// TIA Portal V19 export
FUNCTION_BLOCK "FB21_ManageTowerLight"   // FB21, LAD
{ S7_Optimized_Access := 'TRUE' }
// stored: AutoNumber false, IsIECCheckEnabled true, MemoryReserve 100, SetENOAutomatically false
   VAR_INPUT
      xLightTest { ExternalAccessible := 'False'; ExternalVisible := 'False'; ExternalWritable := 'False'} : Bool;   // Light test
      xConditionReady { ExternalAccessible := 'False'; ExternalVisible := 'False'; ExternalWritable := 'False'} : Bool;   // All condition are Ok
      xStartUpWarning { ExternalAccessible := 'False'; ExternalVisible := 'False'; ExternalWritable := 'False'} : Bool;   // Warning before start
      xReqOpActon { ExternalAccessible := 'False'; ExternalVisible := 'False'; ExternalWritable := 'False'} : Bool;   // Requered Operator action
      xFault { ExternalAccessible := 'False'; ExternalVisible := 'False'; ExternalWritable := 'False'} : Bool;   // Fault or safety
      xPulseSlow { ExternalAccessible := 'False'; ExternalVisible := 'False'; ExternalWritable := 'False'} : Bool;   // Pulse slow
      xPulseFast { ExternalAccessible := 'False'; ExternalVisible := 'False'; ExternalWritable := 'False'} : Bool;   // Pulse fast
   END_VAR
   VAR_OUTPUT
      xGreenLight { ExternalAccessible := 'False'; ExternalVisible := 'False'; ExternalWritable := 'False'} : Bool;   // Tower Green Light
      xOrangeLight { ExternalAccessible := 'False'; ExternalVisible := 'False'; ExternalWritable := 'False'} : Bool;   // Tower Orrange Light
      xRedLight { ExternalAccessible := 'False'; ExternalVisible := 'False'; ExternalWritable := 'False'} : Bool;   // Tower Red Light
      xBuzzer { ExternalAccessible := 'False'; ExternalVisible := 'False'; ExternalWritable := 'False'} : Bool;   // Tower Buzzer
      bCodeRobot { ExternalAccessible := 'False'; ExternalVisible := 'False'; ExternalWritable := 'False'} : Byte;   // Code state for robot
   END_VAR
   VAR
      miDB_TpNewFault { ExternalAccessible := 'False'; ExternalVisible := 'False'; ExternalWritable := 'False'; S7_SetPoint := 'True'} : TP_TIME;
   END_VAR
   VAR_TEMP   // added for the SCL form of the ladder/FBD networks
      _w1 : Bool;
   END_VAR
BEGIN

REGION Network 1: Reset byte code Robot
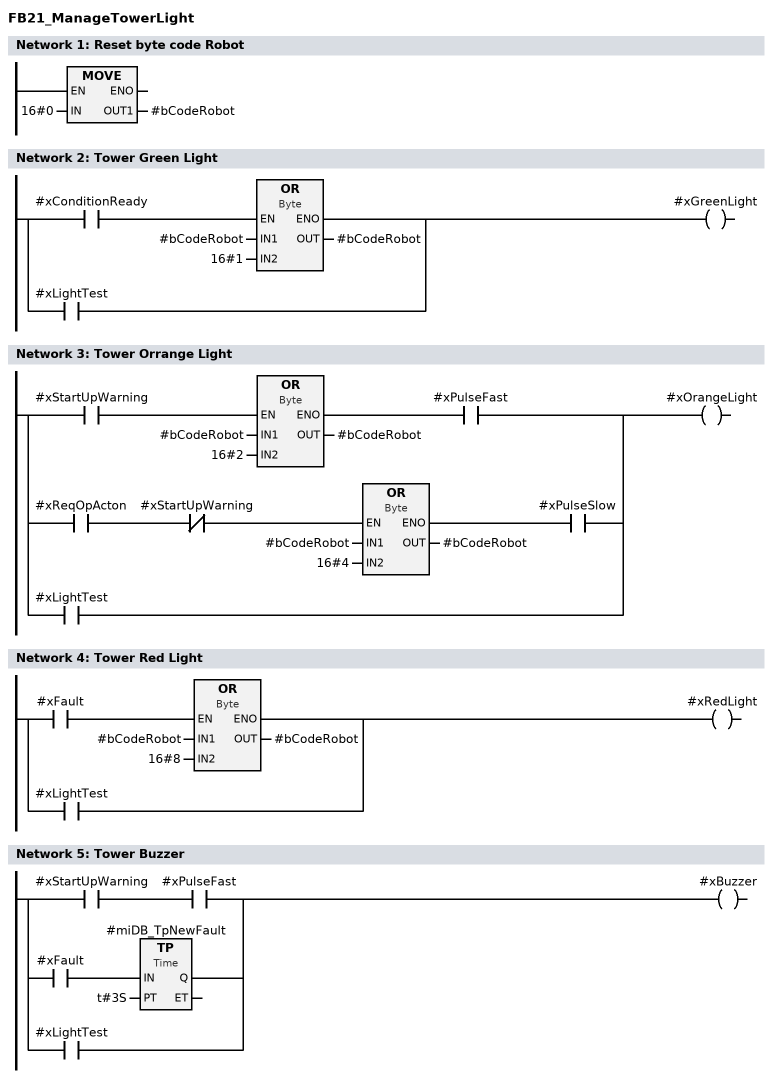
   RUNG wire#powerrail
      Move(in := 16#0, out1 => #bCodeRobot)
   END_RUNG
   // the same network as SCL:
   #bCodeRobot := 16#0;
END_REGION

REGION Network 2: Tower Green Light
   IF #xConditionReady THEN #bCodeRobot := #bCodeRobot OR 16#1; END_IF;
   #xGreenLight := #xConditionReady OR #xLightTest;
END_REGION

REGION Network 3: Tower Orrange Light
   IF #xStartUpWarning THEN #bCodeRobot := #bCodeRobot OR 16#2; END_IF;
   #_w1 := #xReqOpActon AND NOT #xStartUpWarning;
   IF #_w1 THEN #bCodeRobot := #bCodeRobot OR 16#4; END_IF;
   #xOrangeLight := (#xStartUpWarning AND #xPulseFast) OR (#_w1 AND #xPulseSlow) OR #xLightTest;
END_REGION

REGION Network 4: Tower Red Light
   IF #xFault THEN #bCodeRobot := #bCodeRobot OR 16#8; END_IF;
   #xRedLight := #xFault OR #xLightTest;
END_REGION

REGION Network 5: Tower Buzzer
   RUNG wire#powerrail
      Contact( #xStartUpWarning )
      Contact( #xPulseFast )
      wire#w1
      Coil( #xBuzzer )
   END_RUNG
   RUNG wire#powerrail
      Contact( #xFault )
      { S7_Templates := "time_type := Time" } #miDB_TpNewFault.TP(pt := t#3S, et =>)
   END_RUNG wire#w1
   RUNG wire#powerrail
      Contact( #xLightTest )
   END_RUNG wire#w1
   // the same network as SCL:
   #miDB_TpNewFault(IN := #xFault, PT := t#3S);   // TP
   #xBuzzer := (#xStartUpWarning AND #xPulseFast) OR #miDB_TpNewFault.Q OR #xLightTest;
END_REGION
END_FUNCTION_BLOCK
